// TIA Portal project "Project_TestingWIthTurck" (V18)

(* hardware
DEVICE "S7-1500/ET200MP station_1"  S7-1500 station
   slot 0: "Rail_0"  Rack  6ES7 590-1***0-0AA0
   slot 1: "PLC_1"  CPU 1516F-3 PN/DP  6ES7 516-3FN01-0AB0  V2.9
      slot 3: "CPU display_1"  6ES7591-1BA00-0AA0
      slot 32768: "PROFINET interface_1"  X1
      slot 33024: "PROFINET interface_2"  X2
      slot 33280: "DP interface_1"  X3
      slot 34817: "Virtual CP interface port_1"  Virtual CP interface port  Virtual CP interface port
DEVICE "GSD device_1"  GSD.Device.PN
   slot 0: "Rack"  Rack  V1.0
   slot 0: "turck-tbpn-l1-fdio1-2iol"  TBPN-L1-FDIO1-2IOL  6814053  SW V 1.7.35
      slot 0: "DAP v3.1"  DAP v3.1
      slot 1: "PN-IO"  PN-IO
         slot 1: "Port 1"  Port 1
         slot 2: "Port 2"  Port 2
      slot 1: "DXP_1"  DXP
         slot 0: "DXP"  DXP
      slot 2: "PROFIsafe-module_1"  PROFIsafe-module  1.0
         slot 0: "PROFIsafe-module"  PROFIsafe-module
   slot 3: "Safety status_1"  Safety status
      slot 0: "Safety status"  Safety status
   slot 4: "IN 4 WORD/OUT 1 WORD_1"  IN 4 WORD/OUT 1 WORD
      slot 0: "IN 4 WORD/OUT 1 WORD"  IN 4 WORD/OUT 1 WORD
   slot 5: "DI_1"  DI
      slot 0: "DI"  DI
   slot 6: "Diagnostics_1"  Diagnostics
      slot 0: "Diagnostics"  Diagnostics
   slot 7: "IO-Link Events_1"  IO-Link Events
      slot 0: "IO-Link Events"  IO-Link Events
   slot 8: "Module status_1"  Module status
      slot 0: "Module status"  Module status
*)

// ===== PLC "PLC_1"  CPU 1516F-3 PN/DP =====

VAR_GLOBAL   // PLC tag table "Default tag table"
   "Tag_1" AT %M0.0 : Bool;
END_VAR

VAR_GLOBAL   // PLC tag table "Tag table_1"
   "inDXP" AT %I0.0 : "DUT_Array_4bytes";
   "outDXP" AT %Q0.0 : "DUT_Array_2bytes";
   "inSafetyData" AT %I4.0 : "sDUT_Array_2bytes";
   "outSafetyData" AT %Q4.0 : "sDUT_Array_2bytes";
   "inModuleStatus" AT %I112.0 : "DUT_Array_2bytes";
   "inDiagnostics" AT %I40.0 : "DUT_Array_8bytes";
   "inIOLinkEvents" AT %I48.0 : "DUT_Array_64bytes";
   "inSafetyStatus" AT %I10.0 : "DUT_Array_14bytes";
END_VAR

TYPE "DUT_Array_4bytes"
   STRUCT
      raw : Array[0..3] of Byte;
   END_STRUCT;
END_TYPE

TYPE "DUT_Array_2bytes"
   STRUCT
      raw : Array[0..1] of Byte;
   END_STRUCT;
END_TYPE

TYPE "DUT_Array_6bytes"
   STRUCT
      raw : Array[0..5] of Byte;
   END_STRUCT;
END_TYPE

TYPE "sDUT_Array_2bytes"
   STRUCT
      s00_0 : Bool;
      s00_1 : Bool;
      s00_2 : Bool;
      s00_3 : Bool;
      s00_4 : Bool;
      s00_5 : Bool;
      s00_6 : Bool;
      s00_7 : Bool;
      s01_0 : Bool;
      s01_1 : Bool;
      s01_2 : Bool;
      s01_3 : Bool;
      s01_4 : Bool;
      s01_5 : Bool;
      s01_6 : Bool;
      s01_7 : Bool;
   END_STRUCT;
END_TYPE

TYPE "DUT_SafetyStatus_SafetyUnit"
   STRUCT
      SUPM : Bool;   // Safe Unit Protective Mode
      SUCM : Bool;   // Safe Unit Configuration Mode
      SUMM : Bool;   // Safe Unit Unknown Mode
      FBO : Array[0..7] of Bool;
   END_STRUCT;
END_TYPE

TYPE "DUT_ProfiSAFE_StatusByte"
   STRUCT
      iPar_OK : Bool := false;   // The bit is set if new parameter values have been assigned to TBPN-L…-
      DeviceError : Bool := false;   // The bit is set by the device for at least two message cycles if there is amalfunction in the TBPN-L…-FDIO1-2IOL.
      CE_CRC : Bool := false;   // The bit is set if the TBPN-L…-FDIO1-2IOL detects a communication er-ror (CRC error).
      WDTimeout : Bool := false;   // The bit is set if the TBPN-L…-FDIO1-2IOL detects an F communicationerror
      FV_Activated : Bool := false;   // This bit is set during a device restart and in case of an communicationerror.
      Toggle_d : Bool := false;
      Cons_nr_R : Bool := false;   // The bit is set if the TBPN-L…-FDIO1-2IOL the device has reset itscounter for consecutive numbers (Vconsnr_h).
   END_STRUCT;
END_TYPE

TYPE "DUT_diagnostic"
   STRUCT
      VERRV1K89 : Bool;   // Overcurrent sensor supply
      VERRV1K1011 : Bool;   // Overcurrent sensor supply
      VERRV1K1213 : Bool;   // Overcurrent sensor supply
      SCO8 : Bool;   // Overcurrent output
      SCO9 : Bool;   // Overcurrent output
      SCO10 : Bool;   // Overcurrent output
      SCO11 : Bool;   // Overcurrent output
   END_STRUCT;
END_TYPE

TYPE "DUT_IOLINKEVENT"
   STRUCT
      Qualifier : Byte;
      Port : Byte;
      EventCodeH : Byte;
      EventCodeL : Byte;
   END_STRUCT;
END_TYPE

TYPE "DUT_TBPN_L1_Datas"
   STRUCT
      SafetyStatus : "DUT_SafetyStatus";
      Dignostic : "DUT_diagnostic";
      IOLinkEvent : Array[0..15] of "DUT_IOLINKEVENT";
   END_STRUCT;
END_TYPE

TYPE "DUT_Array_8bytes"
   STRUCT
      raw : Array[0..7] of Byte;
   END_STRUCT;
END_TYPE

TYPE "DUT_Array_64bytes"
   STRUCT
      raw : Array[0..63] of Byte;
   END_STRUCT;
END_TYPE

TYPE "DUT_Array_14bytes"
   STRUCT
      raw : Array[0..13] of Byte;
   END_STRUCT;
END_TYPE

TYPE "sDUT_Array_1bytes"
   STRUCT
      s00_0 : Bool;
      s00_1 : Bool;
      s00_2 : Bool;
      s00_3 : Bool;
      s00_4 : Bool;
      s00_5 : Bool;
      s00_6 : Bool;
      s00_7 : Bool;
   END_STRUCT;
END_TYPE

TYPE "DUT_SafetyStatus_FConfig"
   STRUCT
      PMS : Bool;   // No memory chip plugged
      NCNF : Bool;   // No configuration available
      CNFMM : Bool;   // Configuration mismatch
      COMLO : Bool;   // Communication loss
      FERR : Bool;   // Fatal Error
   END_STRUCT;
END_TYPE

TYPE "DUT_SafetyStatus"
   STRUCT
      SafetyUnit : "DUT_SafetyStatus_SafetyUnit";
      PROFISafeErrorCode : Word;
      FConfig : "DUT_SafetyStatus_FConfig";
      Connectors : Array[0..7] of "DUT_SafetyStatus_Connector";
   END_STRUCT;
END_TYPE

TYPE "DUT_SafetyStatus_Connector"
   STRUCT
      RGG : Bool;   // Normal State
      WAIT : Bool;   // Wait for input signal
      TEST : Bool;   // Test input
      ERRFIN : Bool;   // Error at input
      TCCH0 : Bool;   // Cross-circuit channel 0
      TCCH1 : Bool;   // Cross-circuit channel 1
      OVL : Bool;
   END_STRUCT;
END_TYPE

DATA_BLOCK "Main_Safety_RTG1_DB"   // DB1, F_DB
{ S7_Optimized_Access := 'TRUE' }
NAME : FUSI
VERSION : 0.1
// stored: InstanceOfName Main_Safety_RTG1
"Main_Safety_RTG1"
BEGIN
END_DATA_BLOCK

DATA_BLOCK "FB_TBPN_L1_DB"   // DB2
{ S7_Optimized_Access := 'TRUE' }
VERSION : 0.1
// stored: InstanceOfName FB_TBPN_L1
"FB_TBPN_L1"
BEGIN
END_DATA_BLOCK

DATA_BLOCK "DB_Data"   // DB3
{ S7_Optimized_Access := 'TRUE' }
VERSION : 0.1
   VAR
      FBPN_L1_1 : "DUT_TBPN_L1_Datas";
   END_VAR
BEGIN
END_DATA_BLOCK

FUNCTION_BLOCK "Main_Safety_RTG1"   // FB1, F_LAD
{ S7_Optimized_Access := 'TRUE' }
   VAR
      ACK_GL_Instance : ACK_GL;
   END_VAR
   VAR_TEMP
      LightbarrierTriggerred : Bool;
   END_VAR
   VAR CONSTANT
      sTrue : Bool := True;
   END_VAR
BEGIN

REGION Network 1: 1=Acknowledgment for reintegration
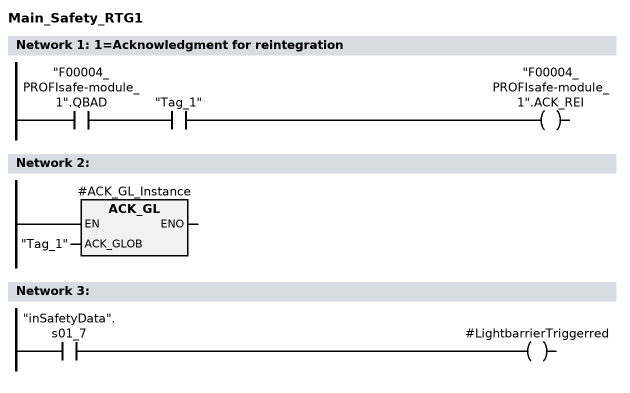
   RUNG wire#powerrail
      Contact( "F00004_PROFIsafe-module_1".QBAD )
      Contact( "Tag_1" )
      Coil( "F00004_PROFIsafe-module_1".ACK_REI )
   END_RUNG
   // the same network as SCL:
   "F00004_PROFIsafe-module_1".ACK_REI := "F00004_PROFIsafe-module_1".QBAD AND "Tag_1";
END_REGION

REGION Network 2
   #ACK_GL_Instance(ACK_GLOB := "Tag_1");   // ACK_GL
END_REGION

REGION Network 3
   RUNG wire#powerrail
      Contact( "inSafetyData".s01_7 )
      Coil( #LightbarrierTriggerred )
   END_RUNG
   // the same network as SCL:
   #LightbarrierTriggerred := "inSafetyData".s01_7;
END_REGION
END_FUNCTION_BLOCK

FUNCTION_BLOCK "FB_TBPN_L1"   // FB2, LAD
{ S7_Optimized_Access := 'TRUE' }
VERSION : 0.1
   VAR_IN_OUT
      ioRawSafetyStatus : Array[*] of Byte;
      ioRawDignostic : Array[*] of Byte;
      ioRawIOLinkEvent : Array[*] of Byte;
      ioData : "DUT_TBPN_L1_Datas";
   END_VAR
   VAR
      SafetyStatus : "FB_TBPN_L1_SafetyStatus";
      Diagnostic : "FB_TBPN_L1_Diagnostic";
      IOLINK_EVENT : "FB_TBPN_L1_IOLinkEvent";
   END_VAR
BEGIN

REGION Network 2
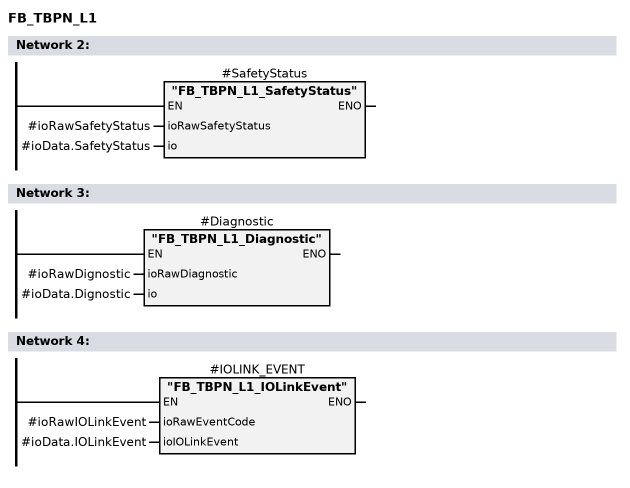
   RUNG wire#powerrail
      #SafetyStatus(ioRawSafetyStatus := #ioRawSafetyStatus, io := #ioData.SafetyStatus)
   END_RUNG
   // the same network as SCL:
   #SafetyStatus(ioRawSafetyStatus := #ioRawSafetyStatus, io := #ioData.SafetyStatus);   // "FB_TBPN_L1_SafetyStatus"
END_REGION

REGION Network 3
   RUNG wire#powerrail
      #Diagnostic(ioRawDiagnostic := #ioRawDignostic, io := #ioData.Dignostic)
   END_RUNG
   // the same network as SCL:
   #Diagnostic(ioRawDiagnostic := #ioRawDignostic, io := #ioData.Dignostic);   // "FB_TBPN_L1_Diagnostic"
END_REGION

REGION Network 4
   RUNG wire#powerrail
      #IOLINK_EVENT(ioRawEventCode := #ioRawIOLinkEvent, ioIOLinkEvent := #ioData.IOLinkEvent)
   END_RUNG
   // the same network as SCL:
   #IOLINK_EVENT(ioRawEventCode := #ioRawIOLinkEvent, ioIOLinkEvent := #ioData.IOLinkEvent);   // "FB_TBPN_L1_IOLinkEvent"
END_REGION
END_FUNCTION_BLOCK

FUNCTION_BLOCK "FB_TBPN_L1_SafetyStatus_SafetyUnit"   // FB3, LAD
{ S7_Optimized_Access := 'TRUE' }
VERSION : 0.1
   VAR_IN_OUT
      ioRawSafetyStatus : Array[*] of Byte;
      io : "DUT_SafetyStatus_SafetyUnit";
   END_VAR
   VAR CONSTANT
      sTure : Bool := True;
   END_VAR
BEGIN

REGION Network 1: Safe Unit Protective Mode
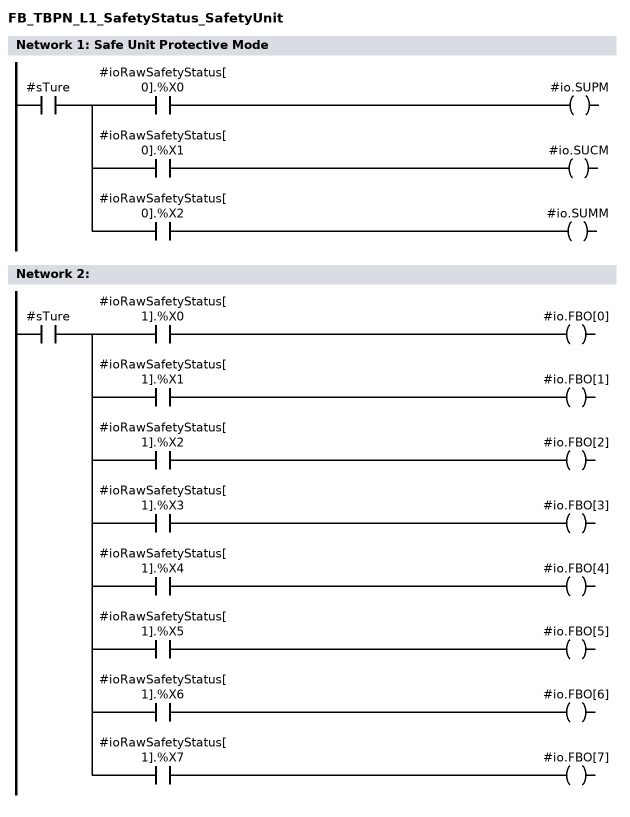
   RUNG wire#powerrail
      Contact( #sTure )
      wire#w1
      Contact( #ioRawSafetyStatus[0].%X0 )
      Coil( #io.SUPM )
   END_RUNG
   RUNG wire#w1
      Contact( #ioRawSafetyStatus[0].%X1 )
      Coil( #io.SUCM )
   END_RUNG
   RUNG wire#w1
      Contact( #ioRawSafetyStatus[0].%X2 )
      Coil( #io.SUMM )
   END_RUNG
   // the same network as SCL:
   #io.SUPM := #sTure AND #ioRawSafetyStatus[0].%X0;
   #io.SUCM := #sTure AND #ioRawSafetyStatus[0].%X1;
   #io.SUMM := #sTure AND #ioRawSafetyStatus[0].%X2;
END_REGION

REGION Network 2
   RUNG wire#powerrail
      Contact( #sTure )
      wire#w1
      Contact( #ioRawSafetyStatus[1].%X0 )
      Coil( #io.FBO[0] )
   END_RUNG
   RUNG wire#w1
      Contact( #ioRawSafetyStatus[1].%X1 )
      Coil( #io.FBO[1] )
   END_RUNG
   RUNG wire#w1
      Contact( #ioRawSafetyStatus[1].%X2 )
      Coil( #io.FBO[2] )
   END_RUNG
   RUNG wire#w1
      Contact( #ioRawSafetyStatus[1].%X3 )
      Coil( #io.FBO[3] )
   END_RUNG
   RUNG wire#w1
      Contact( #ioRawSafetyStatus[1].%X4 )
      Coil( #io.FBO[4] )
   END_RUNG
   RUNG wire#w1
      Contact( #ioRawSafetyStatus[1].%X5 )
      Coil( #io.FBO[5] )
   END_RUNG
   RUNG wire#w1
      Contact( #ioRawSafetyStatus[1].%X6 )
      Coil( #io.FBO[6] )
   END_RUNG
   RUNG wire#w1
      Contact( #ioRawSafetyStatus[1].%X7 )
      Coil( #io.FBO[7] )
   END_RUNG
   // the same network as SCL:
   #io.FBO[0] := #sTure AND #ioRawSafetyStatus[1].%X0;
   #io.FBO[1] := #sTure AND #ioRawSafetyStatus[1].%X1;
   #io.FBO[2] := #sTure AND #ioRawSafetyStatus[1].%X2;
   #io.FBO[3] := #sTure AND #ioRawSafetyStatus[1].%X3;
   #io.FBO[4] := #sTure AND #ioRawSafetyStatus[1].%X4;
   #io.FBO[5] := #sTure AND #ioRawSafetyStatus[1].%X5;
   #io.FBO[6] := #sTure AND #ioRawSafetyStatus[1].%X6;
   #io.FBO[7] := #sTure AND #ioRawSafetyStatus[1].%X7;
END_REGION
END_FUNCTION_BLOCK

FUNCTION_BLOCK "FB_TBPN_L1_SafetyStatus_ProfiSAFEErrorCode"   // FB4, LAD
{ S7_Optimized_Access := 'TRUE' }
VERSION : 0.1
   VAR_IN_OUT
      ioRawSafetyStatus : Array[*] of Byte;
      io : Word;
   END_VAR
   VAR CONSTANT
      sTure : Bool := True;
   END_VAR
BEGIN

REGION Network 1
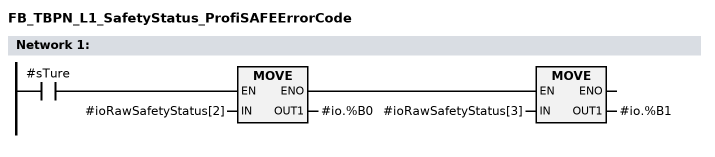
   RUNG wire#powerrail
      Contact( #sTure )
      Move(in := #ioRawSafetyStatus[2], out1 => #io.%B0)
      Move(in := #ioRawSafetyStatus[3], out1 => #io.%B1)
   END_RUNG
   // the same network as SCL:
   IF #sTure THEN
       #io.%B0 := #ioRawSafetyStatus[2];
       #io.%B1 := #ioRawSafetyStatus[3];
   END_IF;
END_REGION
END_FUNCTION_BLOCK

FUNCTION_BLOCK "FB_TBPN_L1_Diagnostic"   // FB5, LAD
{ S7_Optimized_Access := 'TRUE' }
VERSION : 0.1
   VAR_IN_OUT
      ioRawDiagnostic : Array[*] of Byte;
      io : "DUT_diagnostic";
   END_VAR
   VAR CONSTANT
      sTure : Bool := True;
   END_VAR
BEGIN

REGION Network 1: Overcurrent sensor supply
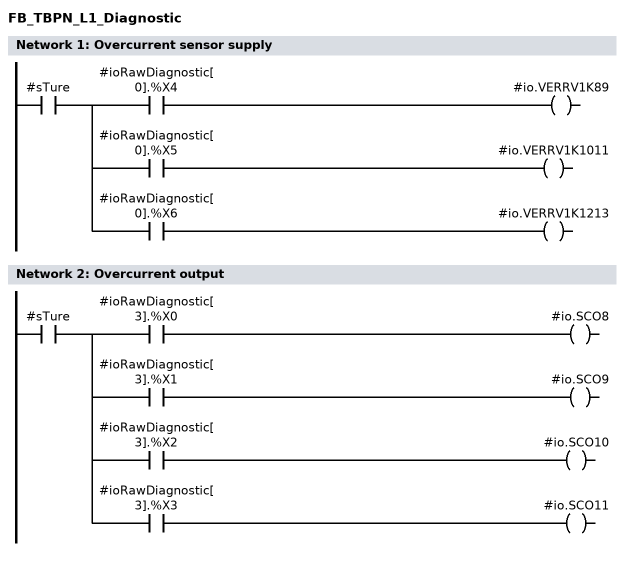
   RUNG wire#powerrail
      Contact( #sTure )
      wire#w1
      Contact( #ioRawDiagnostic[0].%X4 )
      Coil( #io.VERRV1K89 )
   END_RUNG
   RUNG wire#w1
      Contact( #ioRawDiagnostic[0].%X5 )
      Coil( #io.VERRV1K1011 )
   END_RUNG
   RUNG wire#w1
      Contact( #ioRawDiagnostic[0].%X6 )
      Coil( #io.VERRV1K1213 )
   END_RUNG
   // the same network as SCL:
   #io.VERRV1K89 := #sTure AND #ioRawDiagnostic[0].%X4;
   #io.VERRV1K1011 := #sTure AND #ioRawDiagnostic[0].%X5;
   #io.VERRV1K1213 := #sTure AND #ioRawDiagnostic[0].%X6;
END_REGION

REGION Network 2: Overcurrent output
   RUNG wire#powerrail
      Contact( #sTure )
      wire#w1
      Contact( #ioRawDiagnostic[3].%X0 )
      Coil( #io.SCO8 )
   END_RUNG
   RUNG wire#w1
      Contact( #ioRawDiagnostic[3].%X1 )
      Coil( #io.SCO9 )
   END_RUNG
   RUNG wire#w1
      Contact( #ioRawDiagnostic[3].%X2 )
      Coil( #io.SCO10 )
   END_RUNG
   RUNG wire#w1
      Contact( #ioRawDiagnostic[3].%X3 )
      Coil( #io.SCO11 )
   END_RUNG
   // the same network as SCL:
   #io.SCO8 := #sTure AND #ioRawDiagnostic[3].%X0;
   #io.SCO9 := #sTure AND #ioRawDiagnostic[3].%X1;
   #io.SCO10 := #sTure AND #ioRawDiagnostic[3].%X2;
   #io.SCO11 := #sTure AND #ioRawDiagnostic[3].%X3;
END_REGION
END_FUNCTION_BLOCK

FUNCTION_BLOCK "FB_TBPN_L1_IOLinkEvent"   // FB6, LAD
{ S7_Optimized_Access := 'TRUE' }
VERSION : 0.1
   VAR_IN_OUT
      ioRawEventCode : Array[*] of Byte;
      ioIOLinkEvent : Array[0..15] of "DUT_IOLINKEVENT";
   END_VAR
   VAR_TEMP
      i : Int;
   END_VAR
BEGIN

REGION Network 2 (SCL)
   FOR #i := 0 TO 15 DO

       #ioRawEventCode[#i * 4] := #ioIOLinkEvent[#i].Qualifier;
       #ioRawEventCode[#i * 4 + 1] := #ioIOLinkEvent[#i]."Port";
       #ioRawEventCode[#i * 4 + 2] := #ioIOLinkEvent[#i].EventCodeH;
       #ioRawEventCode[#i * 4 + 3] := #ioIOLinkEvent[#i].EventCodeL;
   END_FOR;
END_REGION
END_FUNCTION_BLOCK

FUNCTION_BLOCK "FB_TBPN_L1_SafetyStatus"   // FB7, LAD
{ S7_Optimized_Access := 'TRUE' }
VERSION : 0.1
   VAR_IN_OUT
      ioRawSafetyStatus : Array[*] of Byte;
      io : "DUT_SafetyStatus";
   END_VAR
   VAR
      SafetyUnit : "FB_TBPN_L1_SafetyStatus_SafetyUnit";
      SafetyStatus_ProfiSAFEErrorCode : "FB_TBPN_L1_SafetyStatus_ProfiSAFEErrorCode";
      FConfig : "FB_TBPN_L1_SafetyStatus_FConfig";
      Connectors : Array[0..7] of "FB_TBPN_L1_SafetyStatus_Connector";
   END_VAR
   VAR_TEMP   // added for the SCL form of the ladder/FBD networks
      _w1 : Bool;
   END_VAR
BEGIN

REGION Network 2
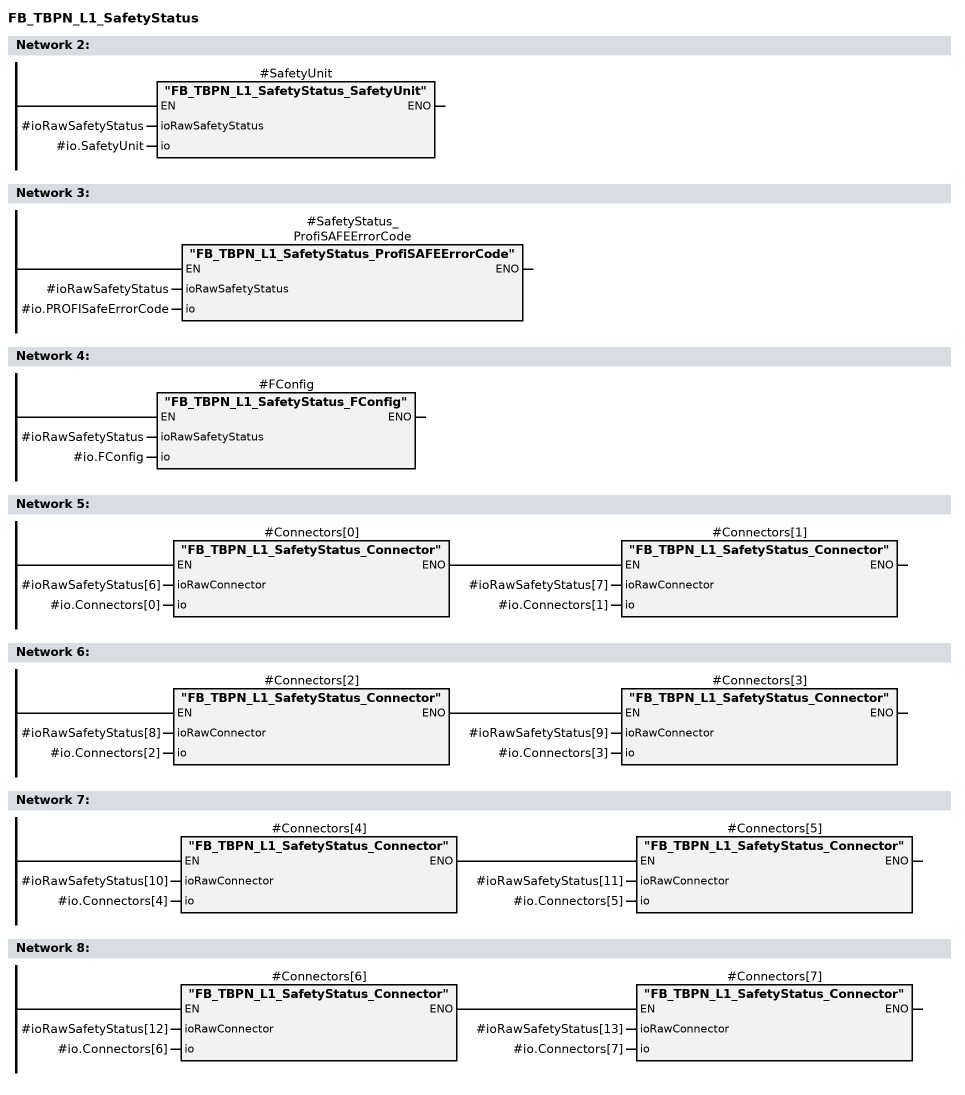
   RUNG wire#powerrail
      #SafetyUnit(ioRawSafetyStatus := #ioRawSafetyStatus, io := #io.SafetyUnit)
   END_RUNG
   // the same network as SCL:
   #SafetyUnit(ioRawSafetyStatus := #ioRawSafetyStatus, io := #io.SafetyUnit);   // "FB_TBPN_L1_SafetyStatus_SafetyUnit"
END_REGION

REGION Network 3
   RUNG wire#powerrail
      #SafetyStatus_ProfiSAFEErrorCode(ioRawSafetyStatus := #ioRawSafetyStatus, io := #io.PROFISafeErrorCode)
   END_RUNG
   // the same network as SCL:
   #SafetyStatus_ProfiSAFEErrorCode(ioRawSafetyStatus := #ioRawSafetyStatus, io := #io.PROFISafeErrorCode);   // "FB_TBPN_L1_SafetyStatus_ProfiSAFEErrorCode"
END_REGION

REGION Network 4
   RUNG wire#powerrail
      #FConfig(ioRawSafetyStatus := #ioRawSafetyStatus, io := #io.FConfig)
   END_RUNG
   // the same network as SCL:
   #FConfig(ioRawSafetyStatus := #ioRawSafetyStatus, io := #io.FConfig);   // "FB_TBPN_L1_SafetyStatus_FConfig"
END_REGION

REGION Network 5
   RUNG wire#powerrail
      #Connectors[0](ioRawConnector := #ioRawSafetyStatus[6], io := #io.Connectors[0])
      #Connectors[1](ioRawConnector := #ioRawSafetyStatus[7], io := #io.Connectors[1])
   END_RUNG
   // the same network as SCL:
   #Connectors[0](ioRawConnector := #ioRawSafetyStatus[6], io := #io.Connectors[0], ENO => #_w1);   // "FB_TBPN_L1_SafetyStatus_Connector"
   IF #_w1 THEN
       #Connectors[1](ioRawConnector := #ioRawSafetyStatus[7], io := #io.Connectors[1]);   // "FB_TBPN_L1_SafetyStatus_Connector"
   END_IF;
END_REGION

REGION Network 6
   RUNG wire#powerrail
      #Connectors[2](ioRawConnector := #ioRawSafetyStatus[8], io := #io.Connectors[2])
      #Connectors[3](ioRawConnector := #ioRawSafetyStatus[9], io := #io.Connectors[3])
   END_RUNG
   // the same network as SCL:
   #Connectors[2](ioRawConnector := #ioRawSafetyStatus[8], io := #io.Connectors[2], ENO => #_w1);   // "FB_TBPN_L1_SafetyStatus_Connector"
   IF #_w1 THEN
       #Connectors[3](ioRawConnector := #ioRawSafetyStatus[9], io := #io.Connectors[3]);   // "FB_TBPN_L1_SafetyStatus_Connector"
   END_IF;
END_REGION

REGION Network 7
   RUNG wire#powerrail
      #Connectors[4](ioRawConnector := #ioRawSafetyStatus[10], io := #io.Connectors[4])
      #Connectors[5](ioRawConnector := #ioRawSafetyStatus[11], io := #io.Connectors[5])
   END_RUNG
   // the same network as SCL:
   #Connectors[4](ioRawConnector := #ioRawSafetyStatus[10], io := #io.Connectors[4], ENO => #_w1);   // "FB_TBPN_L1_SafetyStatus_Connector"
   IF #_w1 THEN
       #Connectors[5](ioRawConnector := #ioRawSafetyStatus[11], io := #io.Connectors[5]);   // "FB_TBPN_L1_SafetyStatus_Connector"
   END_IF;
END_REGION

REGION Network 8
   RUNG wire#powerrail
      #Connectors[6](ioRawConnector := #ioRawSafetyStatus[12], io := #io.Connectors[6])
      #Connectors[7](ioRawConnector := #ioRawSafetyStatus[13], io := #io.Connectors[7])
   END_RUNG
   // the same network as SCL:
   #Connectors[6](ioRawConnector := #ioRawSafetyStatus[12], io := #io.Connectors[6], ENO => #_w1);   // "FB_TBPN_L1_SafetyStatus_Connector"
   IF #_w1 THEN
       #Connectors[7](ioRawConnector := #ioRawSafetyStatus[13], io := #io.Connectors[7]);   // "FB_TBPN_L1_SafetyStatus_Connector"
   END_IF;
END_REGION
END_FUNCTION_BLOCK

FUNCTION_BLOCK "FB_TBPN_L1_SafetyStatus_Connector"   // FB8, LAD
{ S7_Optimized_Access := 'TRUE' }
VERSION : 0.1
   VAR_IN_OUT
      ioRawConnector : Byte;
      io : "DUT_SafetyStatus_Connector";
   END_VAR
   VAR CONSTANT
      sTure : Bool := True;
   END_VAR
BEGIN

REGION Network 1: Normal State
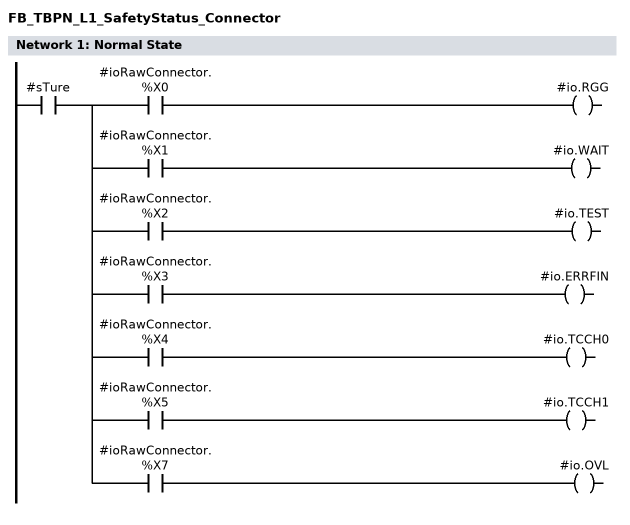
   RUNG wire#powerrail
      Contact( #sTure )
      wire#w1
      Contact( #ioRawConnector.%X0 )
      Coil( #io.RGG )
   END_RUNG
   RUNG wire#w1
      Contact( #ioRawConnector.%X1 )
      Coil( #io.WAIT )
   END_RUNG
   RUNG wire#w1
      Contact( #ioRawConnector.%X2 )
      Coil( #io.TEST )
   END_RUNG
   RUNG wire#w1
      Contact( #ioRawConnector.%X3 )
      Coil( #io.ERRFIN )
   END_RUNG
   RUNG wire#w1
      Contact( #ioRawConnector.%X4 )
      Coil( #io.TCCH0 )
   END_RUNG
   RUNG wire#w1
      Contact( #ioRawConnector.%X5 )
      Coil( #io.TCCH1 )
   END_RUNG
   RUNG wire#w1
      Contact( #ioRawConnector.%X7 )
      Coil( #io.OVL )
   END_RUNG
   // the same network as SCL:
   #io.RGG := #sTure AND #ioRawConnector.%X0;
   #io.WAIT := #sTure AND #ioRawConnector.%X1;
   #io.TEST := #sTure AND #ioRawConnector.%X2;
   #io.ERRFIN := #sTure AND #ioRawConnector.%X3;
   #io.TCCH0 := #sTure AND #ioRawConnector.%X4;
   #io.TCCH1 := #sTure AND #ioRawConnector.%X5;
   #io.OVL := #sTure AND #ioRawConnector.%X7;
END_REGION
END_FUNCTION_BLOCK

FUNCTION_BLOCK "FB_TBPN_L1_SafetyStatus_FConfig"   // FB9, LAD
{ S7_Optimized_Access := 'TRUE' }
VERSION : 0.1
   VAR_IN_OUT
      ioRawSafetyStatus : Array[*] of Byte;
      io : "DUT_SafetyStatus_FConfig";
   END_VAR
   VAR CONSTANT
      sTure : Bool := True;
   END_VAR
BEGIN

REGION Network 1: No memory chip plugged
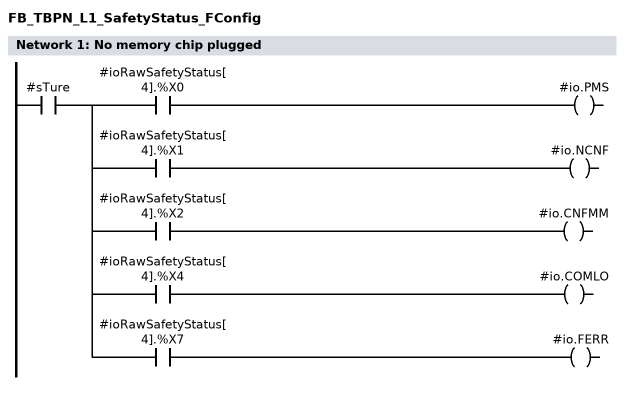
   RUNG wire#powerrail
      Contact( #sTure )
      wire#w1
      Contact( #ioRawSafetyStatus[4].%X0 )
      Coil( #io.PMS )
   END_RUNG
   RUNG wire#w1
      Contact( #ioRawSafetyStatus[4].%X1 )
      Coil( #io.NCNF )
   END_RUNG
   RUNG wire#w1
      Contact( #ioRawSafetyStatus[4].%X2 )
      Coil( #io.CNFMM )
   END_RUNG
   RUNG wire#w1
      Contact( #ioRawSafetyStatus[4].%X4 )
      Coil( #io.COMLO )
   END_RUNG
   RUNG wire#w1
      Contact( #ioRawSafetyStatus[4].%X7 )
      Coil( #io.FERR )
   END_RUNG
   // the same network as SCL:
   #io.PMS := #sTure AND #ioRawSafetyStatus[4].%X0;
   #io.NCNF := #sTure AND #ioRawSafetyStatus[4].%X1;
   #io.CNFMM := #sTure AND #ioRawSafetyStatus[4].%X2;
   #io.COMLO := #sTure AND #ioRawSafetyStatus[4].%X4;
   #io.FERR := #sTure AND #ioRawSafetyStatus[4].%X7;
END_REGION
END_FUNCTION_BLOCK

ORGANIZATION_BLOCK "Main"   // OB1, LAD, ProgramCycle
TITLE = "Main Program Sweep (Cycle)"
{ S7_Optimized_Access := 'TRUE' }
VERSION : 0.1
   VAR_INPUT
      Initial_Call : Bool;   // Initial call of this OB
      Remanence : Bool;   // =True, if remanent data are available
   END_VAR
   VAR_TEMP
      FieldbusBit00_07 : Bool;
   END_VAR
BEGIN

REGION Network 2
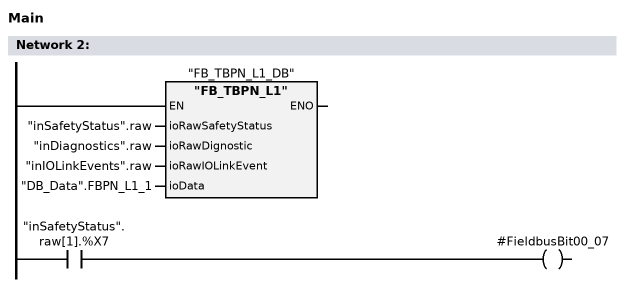
   RUNG wire#powerrail
      "FB_TBPN_L1_DB"(ioRawSafetyStatus := "inSafetyStatus".raw, ioRawDignostic := "inDiagnostics".raw, ioRawIOLinkEvent := "inIOLinkEvents".raw, ioData := "DB_Data".FBPN_L1_1)
   END_RUNG
   RUNG wire#powerrail
      Contact( "inSafetyStatus".raw[1].%X7 )
      Coil( #FieldbusBit00_07 )
   END_RUNG
   // the same network as SCL:
   "FB_TBPN_L1_DB"(ioRawSafetyStatus := "inSafetyStatus".raw,   // "FB_TBPN_L1"
                   ioRawDignostic := "inDiagnostics".raw,
                   ioRawIOLinkEvent := "inIOLinkEvents".raw,
                   ioData := "DB_Data".FBPN_L1_1);
   #FieldbusBit00_07 := "inSafetyStatus".raw[1].%X7;
END_REGION
END_ORGANIZATION_BLOCK